FUNCTION "LnkJ_FixtureCmd" : Void
{ S7_Optimized_Access := 'TRUE' }
VERSION : 0.1
   VAR_INPUT
      Seq : UInt;   // 엔벨로프 seq (1..65535, 0 = 없음)
   END_VAR

   VAR_IN_OUT
      Buf : Array[*] of Byte;   // 출력 버퍼
      Pos : DInt;   // 다음 쓸 절대 인덱스 (< 0 = 오류 유지)
      Val : "LNK_FixtureSub";   // data
   END_VAR


BEGIN
	// GENERATED by gr-contract gen-link from message "FixtureCmd" (id 41, "LNK_FixtureSub" sig 16#AFBB75A6) - do not edit
	// {"type":"FixtureCmd","seq":<Seq>,"sig":2948298150,"data":<Val>}
	"Json_WRaw"(Buf := #Buf, Pos := #Pos, Lit := '{"type":"FixtureCmd","seq":');
	"Json_WUInt"(Buf := #Buf, Pos := #Pos, Val := #Seq);
	"Json_WRaw"(Buf := #Buf, Pos := #Pos, Lit := ',"sig":2948298150,"data":');
	"JsonW_LNK_FixtureSub"(Buf := #Buf, Pos := #Pos, Val := #Val);
	"Json_WRaw"(Buf := #Buf, Pos := #Pos, Lit := '}');
END_FUNCTION
